{attribute 'GeneratedUsingTerminal: IODEVICETYPE_ETHERCATPROT'}
{attribute addProperty BoxType "IODEVICETYPE_ETHERCATPROT"}
{attribute addProperty Id "Beckhoff_EP1xxxBeckhoff_EP1xxx_D62248F51572Beckhoff_EP2xxxBeckhoff_EP2xxx_268196C73266Beckhoff_EP3xxxBeckhoff_EP3xxx_3EBBF4AC2708Beckhoff_EP4xxxBeckhoff_EP4xxx_BBA678B0256Beckhoff_EP5xxxBeckhoff_EP5xxx_0672B834313Beckhoff_EP6xxxBeckhoff_EP6xxx_2F08A32E1118Beckhoff_EP7xxxBeckhoff_EP7xxx_B925E5352560Beckhoff_EP8xxxBeckhoff_EP8xxx_337C41A0250Beckhoff_EP9xxxBeckhoff_EP9xxx_3941D599561SyncUnitsSyncUnits_2E61B95536InputsInputs_25A0042B160OutputsOutputs_2397A10E106InfoDataInfoData_C76BEFB322"}
{attribute addProperty CRC "4193554618"}
{attribute addProperty Size "12928"}
TYPE EtherCAT_Master_EPxxxx_F9F490BA :
STRUCT
	{attribute addProperty Name "Beckhoff_EP1xxx"}
	{attribute addProperty PreviousPort "EtherCAT_Master_EPxxxx : Master"}
	Beckhoff_EP1xxx : Beckhoff_EP1xxx_D62248F5;
	{attribute addProperty Name "Beckhoff_EP2xxx"}
	{attribute addProperty PreviousPort "Beckhoff EP1xxx : C"}
	Beckhoff_EP2xxx : Beckhoff_EP2xxx_268196C7;
	{attribute addProperty Name "Beckhoff_EP3xxx"}
	{attribute addProperty PreviousPort "Beckhoff EP2xxx : C"}
	Beckhoff_EP3xxx : Beckhoff_EP3xxx_3EBBF4AC;
	{attribute addProperty Name "Beckhoff_EP4xxx"}
	{attribute addProperty PreviousPort "Beckhoff EP3xxx : C"}
	Beckhoff_EP4xxx : Beckhoff_EP4xxx_BBA678B0;
	{attribute addProperty Name "Beckhoff_EP5xxx"}
	{attribute addProperty PreviousPort "Beckhoff EP4xxx : C"}
	Beckhoff_EP5xxx : Beckhoff_EP5xxx_0672B834;
	{attribute addProperty Name "Beckhoff_EP6xxx"}
	{attribute addProperty PreviousPort "Beckhoff EP5xxx : C"}
	Beckhoff_EP6xxx : Beckhoff_EP6xxx_2F08A32E;
	{attribute addProperty Name "Beckhoff_EP7xxx"}
	{attribute addProperty PreviousPort "Beckhoff EP6xxx : C"}
	Beckhoff_EP7xxx : Beckhoff_EP7xxx_B925E535;
	{attribute addProperty Name "Beckhoff_EP8xxx"}
	{attribute addProperty PreviousPort "Beckhoff EP7xxx : C"}
	Beckhoff_EP8xxx : Beckhoff_EP8xxx_337C41A0;
	{attribute addProperty Name "Beckhoff_EP9xxx"}
	{attribute addProperty PreviousPort "Beckhoff EP8xxx : C"}
	Beckhoff_EP9xxx : Beckhoff_EP9xxx_3941D599;
	{attribute addProperty Name "SyncUnits"}
	SyncUnits : SyncUnits_2E61B955;
	{attribute addProperty Name "Inputs"}
	Inputs : Inputs_25A0042B;
	{attribute addProperty Name "Outputs"}
	Outputs : Outputs_2397A10E;
	{attribute addProperty Name "InfoData"}
	InfoData : InfoData_C76BEFB3;
END_STRUCT
END_TYPE

(* stored: Version 1.2.0.0, ProductVersion 3.1.4024.9
   DUT EtherCAT_Master_EPxxxx_F9F490BA: Id {f2769992-98c9-4e52-a89d-a2f66cda2ca8} *)
